(* IEC 61131-3 sources: RL_MAR/experiments/comparison/autoplc/results/gpt-4o_20260511_211137/med_22, 1 file *)

(* ---- med_22_1.st ---- *)
FUNCTION_BLOCK CottonCandyMachine
VAR_INPUT
    SugarLevel : REAL; (* Input for sugar level *)
    SpinningSpeed : INT; (* Input for spinning speed *)
END_VAR
VAR_OUTPUT
    SugarFeeder : BOOL; (* Output to control sugar feeding *)
    MotorSpeed : INT; (* Output to control spinning motor speed *)
END_VAR

VAR
    (* Internal variables can be declared here if needed *)
END_VAR

(* Initialization of output variables *)
SugarFeeder := FALSE;
MotorSpeed := 0;

(* Control logic for sugar feeding mechanism *)
IF SugarLevel < 10.0 THEN
    SugarFeeder := TRUE; (* Activate sugar feeder *)
ELSE
    SugarFeeder := FALSE; (* Deactivate sugar feeder *)
END_IF

(* Control logic for motor speed *)
IF SpinningSpeed > 0 THEN
    MotorSpeed := SpinningSpeed; (* Set motor speed to input spinning speed *)
ELSE
    MotorSpeed := 0; (* Set motor speed to 0 if input speed is 0 or negative *)
END_IF

END_FUNCTION_BLOCK
